# EPICS substitutions: evrSupport/Db/ioc/bsaTOROEdef.substitutions
#==============================================================================
#
# Abs:  Beam Synchronous Acquisition records for a single Toroid.
#
# Name: bsaTOROEdef.substitutions
#
# Note: Must follow the LCLS naming conventions.
#
#==============================================================================
#
file bsaATTREdef.db
{
#           Device  Attribute  Input           EGU       HOPR LOPR PREC ADEL   Link
  pattern {   D       , ATTR , I              , EG     , HO     , LO     , PR     , AD     ,  LNK,     SINK_SIZE    }
	  { $(DEVICE) , TMIT , $(DEVICE):TMIT , $(EGU) , $(HOPR), $(LOPR), $(PREC), $(ADEL),$(SLCLNK),  $(SINK_SIZE\=10) }
}
